Fanuc KAREL source: IO0073.KL

-- PROVISIONAL review KL for V1013-1; original PC SHA256 32ee403f94f4df55f4b5d434dd98f3e494d27d3db9c45a7e1a2f4d101fa798b7
-- Incomplete behavior may be omitted. Consult companion uncertainty JSON. Do not deploy.
PROGRAM IO0073
%NOLOCKGROUP
-- UNRESOLVED_LOCAL_POOL 5 cells at code offset 13; source declarations unknown
-- DIRECT_LOCAL_WORD_ACCESS alone does not prove INTEGER, REAL, or BOOLEAN
BEGIN
  -- UNRESOLVED_PC offsets 0-18; opcodes 2B,2C,7B
  -- UNRESOLVED_PC offsets 23-30; opcodes 9D,23
  -- UNRESOLVED_PC offsets 35-49; opcodes 2E,22,9D,33,35
  -- UNRESOLVED_PC offsets 54-61; opcodes 9D,23
  -- UNRESOLVED_PC offsets 66-77; opcodes 2E,23
  -- UNRESOLVED_PC offsets 82-99; opcodes 21,9D,52,19,9C,5B,79
  -- UNRESOLVED_PC offsets 104-118; opcodes 21,9D,52,23
  -- UNRESOLVED_PC offsets 128-132; opcodes 7F
  -- UNRESOLVED_PC offsets 137-141; opcodes 27,AA
  -- UNRESOLVED_PC offsets 146-150; opcodes 7F
END IO0073
